{attribute 'linkalways'} 
{attribute 'no_explicit_call' := 'This FB is a CLASS and must be accessed using methods or properties'}
{attribute 'enable_dynamic_creation'}
FUNCTION_BLOCK Node_F_VN_SigmoidExp EXTENDS VisionNode
VAR
    ipSrcImage : _ITcVnImage;
    ipDestImage : _ITcVnImage;
    fShift : _REAL(0.0);
    fSteepness : _REAL(0.0);
    hrPrev : _HRESULT(S_OK);
	hresult : _HRESULT(S_OK);
END_VAR

METHOD PUBLIC  Clone : I_Node
VAR
	pNode : POINTER TO Node_F_VN_SigmoidExp;
END_VAR
pNode := __NEW(Node_F_VN_SigmoidExp);
Clone := pNode^;
END_METHOD

METHOD FB_init : BOOL
VAR_INPUT
	bInitRetains : BOOL; // if TRUE, the retain variables are initialized (warm start / cold start)
	bInCopyCode : BOOL;  // if TRUE, the instance afterwards gets moved into the copy code (online change)
END_VAR
AddInput('ipSrcImage', ipSrcImage);
AddParameter('fShift', fShift);
AddParameter('fSteepness', fSteepness);
AddInput('hrPrev', hrPrev);
AddOutput('ipDestImage', ipDestImage);
AddOutput('hresult',hresult);
END_METHOD

METHOD PROTECTED OnExecute
hresult.Value := F_VN_SigmoidExp(
    ipSrcImage := ipSrcImage.Value,
	ipDestImage := ipDestImage.Value,
    fShift := fShift.Value,
    fSteepness := fSteepness.Value,
	hrPrev:= hrPrev.Value);
END_METHOD

METHOD PUBLIC PreExecutionCheck
VAR_INPUT
	Check : I_PreExecutionChecks;
END_VAR
Check.IsTrue(ipSrcImage.IsValid, 'ipSrcImage must contain an image');
Check.IsTrue(ipSrcImage.IsPixelDepth(32), 'ipSrcImage must have 32 bit pixel depth');
END_METHOD

END_FUNCTION_BLOCK

(* stored: Version 1.1.0.1, ProductVersion 3.1.4024.13
   POU Node_F_VN_SigmoidExp: Id {e9da0b28-42d0-0ba0-2597-5cc7adf08197}, SpecialFunc None
   Folder Constructor: Id {b5562c86-7aad-0486-33fd-6523202aee7e}
   Method Clone: Id {c348e51b-c2a6-09a0-3e13-5b5760d04707}
   Method FB_init: Id {c3c3f09e-f5e2-0ad1-1d7b-30e77e92f960}
   Method OnExecute: Id {03f5dd6a-11dd-0402-0232-a7453647a392}
   Method PreExecutionCheck: Id {43a68e4b-22c1-0f77-0ef3-f95c16b44f38} *)
